TYPE ST_EM_Template_Config :
STRUCT
	// Digital inputs
	// n.a.
	
	// Digital outputs
	// n.a.
	
	// Alarms
	// n.a.
	
	// CM's
	// n.a.
	
	// Others
	// n.a.
	
END_STRUCT
END_TYPE

(* stored: Version 1.1.0.1, ProductVersion 3.1.4024.10
   DUT ST_EM_Template_Config: Id {c2b077c5-465a-495c-936c-4e3315cad05c} *)
